{attribute addProperty BoxType "ER3314-0002-0021"}
{attribute addProperty Id "TC_Inputs_ChannelAT %I*ARRAY[0..3] OF TC_Inputs_Channel_F16A160D128160WcStateAT %I*WcState_F855686C1620InfoDataAT %I*InfoData_BC63D37F80100"}
{attribute addProperty CRC "2738248042"}
{attribute addProperty SizeInBites "224"}
{attribute addProperty SizeInBytes "28"}
TYPE ER3314_2E54E3B0 :
STRUCT
	{attribute addProperty Name "TC_Inputs_Channel"}
	TC_Inputs_Channel : ARRAY[0..3] OF TC_Inputs_Channel_F16A160D;
	{attribute addProperty Name "WcState"}
	WcState : WcState_F855686C;
	{attribute addProperty Name "InfoData"}
	InfoData : InfoData_BC63D37F;
END_STRUCT
END_TYPE

(* stored: Version 1.2.0.0, ProductVersion 3.1.4024.9
   DUT ER3314_2E54E3B0: Id {e4166221-2fa0-43d3-ad96-534b89daa349} *)
